TYPE ST_Subscriber :
STRUCT
	nHandle			: UDINT;
	stAdsStatus		: ST_AdsStatus;
	fbRPC			: FB_RPC_Dynamic;
END_STRUCT
END_TYPE

(* stored: Version 1.1.0.1, ProductVersion 3.1.4024.12
   DUT ST_Subscriber: Id {67a39308-d764-4927-baf0-a2373e465972} *)
